FUNCTION_BLOCK MoveLeft EXTENDS GuardMove
VAR_INPUT
END_VAR
VAR_OUTPUT
END_VAR
VAR
END_VAR

(*

short summary
=================
This abstract property returns the class name of the concrete object, 
which is useful for logging/debugging purpose or to check the class name
for ``__DELETE`` in factories (sometimes it's necessary to do more 
than just to free the memory).

.. <legal notes>

legal notes
=================
| SPDX-FileCopyrightText: © 2022 ekvip automation GmbH <info@ekvip.de>
| SPDX-License-Identifier: Apache-2.0
| For details check: Apache-2.0_

.. _Apache-2.0: https://www.apache.org/licenses/LICENSE-2.0

.. </legal notes>

*)
PROPERTY className : CNM_AbstractObject.ClassName
GET
className := 'MoveLeft';
END_GET
END_PROPERTY

PROPERTY PROTECTED direction : Rotation
GET
direction := Rotation.LEFT;
END_GET
END_PROPERTY

END_FUNCTION_BLOCK

(* stored: Version 1.1.0.1
   POU MoveLeft: Id {ea0ec2c9-e0a4-4732-9c3b-d55d6250ff60}, SpecialFunc None
   Property className: Id {8b86d80d-49b2-4159-8a57-7dc9ec9c2cc0}
   Get Get: Id {35d7c351-b97f-491c-a412-01c5c8910b21}
   Property direction: Id {57addffb-ab44-41bf-abe2-004a30218ec3}
   Get Get: Id {cf2cab31-e8d9-4ae2-a598-f9b9c6004612} *)
